FUNCTION_BLOCK Reset6
VAR_INPUT
END_VAR
VAR_OUTPUT
END_VAR
VAR
END_VAR

END_FUNCTION_BLOCK

(* stored: Version 1.1.0.1, ProductVersion 3.1.4024.11
   POU Reset6: Id {948c74cf-5c3d-414a-8f30-2fa391cefd79}, SpecialFunc None *)
